// TIA Portal V17 export
// export: Created 2022-07-20T06:59:39.3716126Z, ExportSetting WithDefaults, DisplayName Totally Integrated Automation Portal, DisplayVersion V17, DisplayName TIA Portal Openness, DisplayVersion V17, DisplayName TIA Portal Version Control Interface, DisplayVersion V17, DisplayName SINAMICS Startdrive Advanced, DisplayVersion V17, DisplayName SINAMICS Startdrive G130, G150, S120, S150, SINAMICS MV, S210, DisplayVersion V17, DisplayName SINAMICS Startdrive G110M, G120, G120C, G120D, G120P, G115D, DisplayVersion V17, DisplayName STEP 7 Professional, DisplayVersion V17, DisplayName STEP 7 Safety, DisplayVersion V17, DisplayName WinCC Advanced, DisplayVersion V17
FUNCTION "FC10014_RealTo2Int" : Void   // FC10014, LAD
TITLE = FC10014_RealTo2Int
{ S7_Optimized_Access := 'TRUE' }
AUTHOR : Anirouddh
FAMILY : 1001x_CONVERT
VERSION : 1.0
// Release note : 
// 1.0 - Feature developped
// stored: AutoNumber false, IsIECCheckEnabled false, SetENOAutomatically false, UDAEnableTagReadback false
   VAR_INPUT
      Real_Input : Real;
   END_VAR
   VAR_OUTPUT
      Int_LowWeight : Int;
      Int_HighWeight : Int;
   END_VAR
   VAR_TEMP
      Val_temp1 : DWord;
   END_VAR
BEGIN

REGION Network 1 (SCL): FC10014_RealTo2Int
   //Entier bits de poids fort
   #Int_LowWeight := REAL_TO_INT(#Real_Input);

   //Entier bits de poids faible
   #Val_temp1 := REAL_TO_DWORD(#Real_Input);

   #Val_temp1 := SHR_DWORD(IN := #Val_temp1, N := 16);

   #Int_HighWeight := DWORD_TO_INT(#Val_temp1);
END_REGION
END_FUNCTION
